# EPICS autosave request: BPMApp/Db/MonitDspCtl_settings.req
$(P)$(R)MonitEnable
